// Mitsubishi GX Works2 project: BookEX6_47 Serial   PLC: Q13UDV

// global labels: Global
VAR_GLOBAL
  bVar0 AT M5000 : BOOL;
  abArray0 AT M5010 : ARRAY [0..49] OF BOOL;
  sStr0 AT D5000 : STRING[199];
  sStr1 AT D5100 : STRING[199];
  sStr2 AT D5200 : STRING[199];
  sStr3 AT D5300 : STRING[199];
  sStr4 AT D5400 : STRING[199];
  sStr5 AT D5500 : STRING[199];
  sStr6 AT D5600 : STRING[199];
  sStr7 AT D5700 : STRING[199];
  sStr8 AT D5800 : STRING[199];
  sStr9 AT D5900 : STRING[199];
  iVar0 AT D4500 : INT;
  iVar1 AT D4501 : INT;
  iVar2 AT D4502 : INT;
  iVar3 AT D4503 : INT;
  iVar4 AT D4504 : INT;
  iVar5 AT D4505 : INT;
  iVar6 AT D4506 : INT;
  iVar7 AT D4507 : INT;
  iVar8 AT D4508 : INT;
  iVar9 AT D4509 : INT;
  dVar0 AT D4510 : DINT;
  dVar1 AT D4512 : DINT;
  dVar2 AT D4514 : DINT;
  dVar3 AT D4516 : DINT;
  dVar4 AT D4518 : DINT;
  dVar5 AT D4520 : DINT;
  dVar6 AT D4522 : DINT;
  dVar7 AT D4524 : DINT;
  dVar8 AT D4526 : DINT;
  dVar9 AT D4528 : DINT;
  wVar0 AT D4530 : WORD;
  wVar1 AT D4531 : WORD;
  wVar2 AT D4532 : WORD;
  wVar3 AT D4533 : WORD;
  wVar4 AT D4534 : WORD;
  wVar5 AT D4535 : WORD;
  wVar6 AT D4536 : WORD;
  wVar7 AT D4537 : WORD;
  wVar8 AT D4538 : WORD;
  wVar9 AT D4539 : WORD;
  dwVar0 AT D4540 : DWORD;
  dwVar1 AT D4542 : DWORD;
  dwVar2 AT D4544 : DWORD;
  dwVar3 AT D4546 : DWORD;
  dwVar4 AT D4548 : DWORD;
  dwVar5 AT D4550 : DWORD;
  dwVar6 AT D4552 : DWORD;
  dwVar7 AT D4554 : DWORD;
  dwVar8 AT D4556 : DWORD;
  dwVar9 AT D4558 : DWORD;
  fsVar0 AT D4560 : REAL;
  fsVar1 AT D4562 : REAL;
  fsVar2 AT D4564 : REAL;
  fsVar3 AT D4566 : REAL;
  fsVar4 AT D4568 : REAL;
  fsVar5 AT D4570 : REAL;
  fsVar6 AT D4572 : REAL;
  fsVar7 AT D4574 : REAL;
  fsVar8 AT D4576 : REAL;
  fsVar9 AT D4578 : REAL;
  fdVar0 AT D4580 : LREAL;
  tTime0 AT D4620 : TIME;
  tTime1 AT D4622 : TIME;
  tTime2 AT D4624 : TIME;
  tTime3 AT D4626 : TIME;
  tTime4 AT D4628 : TIME;
  tTime5 AT D4630 : TIME;
  tTime6 AT D4632 : TIME;
  tTime7 AT D4634 : TIME;
  tTime8 AT D4636 : TIME;
  tTime9 AT D4638 : TIME;
  tTime10 AT D4640 : TIME;
  bVar1 AT M5001 : BOOL;
  bVar2 AT M5002 : BOOL;
  bVar3 AT M5003 : BOOL;
  bVar4 AT M5004 : BOOL;
  bVar5 AT M5005 : BOOL;
  bVar6 AT M5006 : BOOL;
  bVar7 AT M5007 : BOOL;
  bVar8 AT M5008 : BOOL;
  bVar9 AT M5009 : BOOL;
  abArray1 AT M5060 : ARRAY [0..49] OF BOOL;
  abArray2 AT M5110 : ARRAY [0..49] OF BOOL;
  abArray3 AT M5160 : ARRAY [0..49] OF BOOL;
  abArray4 AT M5210 : ARRAY [0..49] OF BOOL;
  abArray5 AT M5260 : ARRAY [0..49] OF BOOL;
  abArray6 AT M5310 : ARRAY [0..49] OF BOOL;
  abArray7 AT M5360 : ARRAY [0..49] OF BOOL;
  abArray8 AT M5410 : ARRAY [0..49] OF BOOL;
  abArray9 AT M5460 : ARRAY [0..49] OF BOOL;
  fdVar1 AT D4584 : LREAL;
  fdVar2 AT D4588 : LREAL;
  fdVar3 AT D4592 : LREAL;
  fdVar4 AT D4596 : LREAL;
  fdVar5 AT D4600 : LREAL;
  fdVar6 AT D4604 : LREAL;
  fdVar7 AT D4608 : LREAL;
  fdVar8 AT D4612 : LREAL;
  fdVar9 AT D4616 : LREAL;
  afsPen0 AT D2000 : ARRAY [0..499] OF REAL;
  afsPen1 AT D3000 : ARRAY [0..499] OF REAL;
  adwD10 AT D10 : ARRAY [0..9] OF DWORD;
  awD10 AT D10 : ARRAY [0..19] OF WORD;
  abM10 AT M10 : ARRAY [0..19] OF BOOL;
END_VAR

// global labels: CommVar
VAR_GLOBAL
  CommRx AT D100 : ARRAY [0..49] OF INT;
  CommTx AT D300 : ARRAY [0..49] OF INT;
  gbNormal AT M10 : BOOL;
  gbError AT M11 : BOOL;
  giErrCnt AT D12 : INT;
  giOKCnt AT D13 : INT;
END_VAR
// user libraries (not included): HMI

FUNCTION_BLOCK BattRequest
VAR_INPUT
  b_EN : BOOL;
END_VAR
VAR_OUTPUT
  b_ENO : BOOL;
END_VAR
VAR
  ix : INT;
  iy : INT;
  iz : INT;
END_VAR
;
b_ENO := b_EN;
IF b_EN THEN
	CommTX[0] := 11;
	CommTX[1] := HFAAF;
	CommTx[2] := H0560;
	CommTx[3] := H6001;
	CommTx[4] := H0047;
	CommTx[5] := HAF00;
	CommTx[6] := H00A0;
	iy := 0;
	FOR ix := 2 TO 4 DO
		iz := CommTx[ix] MOD 256;
		iy := iy + iz;
		iz := CommTx[ix] / 256;
		iy := iy + iz;
	END_FOR;
	CommTx[5] := CommTx[5] + (iy MOD 256);	
END_IF;
END_FUNCTION_BLOCK

FUNCTION_BLOCK BattStatus
VAR_INPUT
  b_EN : BOOL;
END_VAR
VAR_OUTPUT
  b_ENO : BOOL;
END_VAR
VAR
  ix : INT;
END_VAR
;
b_ENO := b_EN;
IF b_EN THEN
	ix := CommRx[4];
	SWAP(TRUE, ix);
	fsVar0 := INT_TO_REAL(ix) / 100.0;
	ix := CommRx[5];
	SWAP(TRUE, ix);
	fsVar1 := INT_TO_REAL(ix) / 100.0;
	ix := CommRx[6];
	SWAP(TRUE, ix);
	fsVar2 := INT_TO_REAL(ix);
	ix := CommRx[7];
	SWAP(TRUE, ix);
	fsVar3 := INT_TO_REAL(ix) / 10.0;
END_IF;
END_FUNCTION_BLOCK

PROGRAM ExBARCODE
(* structured ladder/FBD written out as ST: instructions are called as NAME(EN, inputs, outputs); _pN, _eN, _tN stand for wires *)
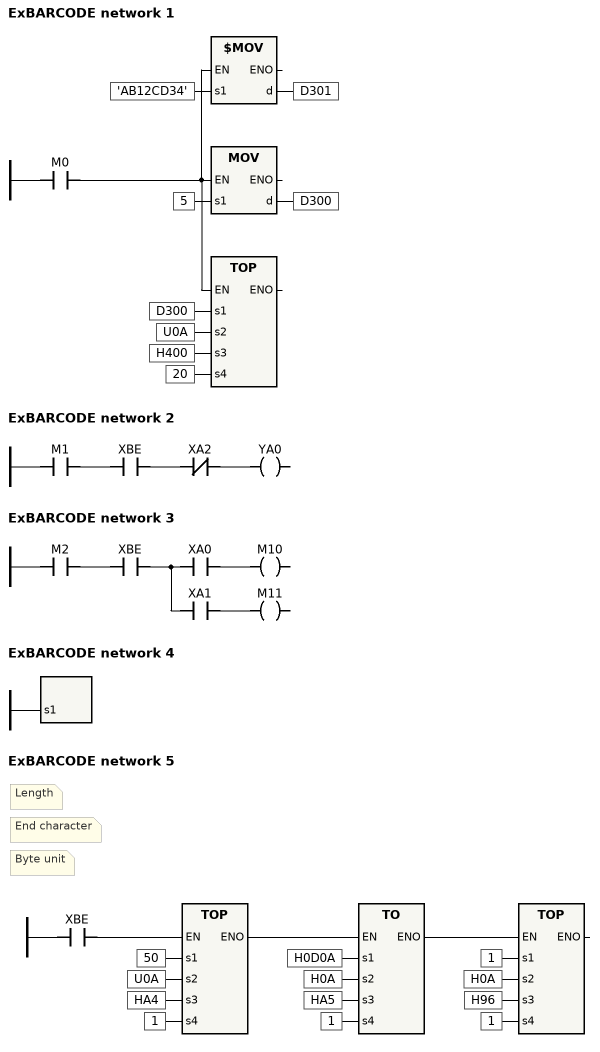
(* network 1 *)
$MOV(M0, 'AB12CD34', D301);
MOV(M0, 5, D300);
TOP(M0, D300, U0A, H400, 20);
(* network 2 *)
YA0 := M1 AND XBE AND NOT XA2;
(* network 3 *)
_p1 := M2 AND XBE;
M10 := _p1 AND XA0;
M11 := _p1 AND XA1;
(* network 4 *)
(* element kind 10  <- TRUE *)
(* network 5 *)
(* Length *)
(* End character *)
(* Byte unit *)
_e1 := TOP(XBE, 50, U0A, HA4, 1);
_e2 := TO(_e1, H0D0A, H0A, HA5, 1);
TOP(_e2, 1, H0A, H96, 1);
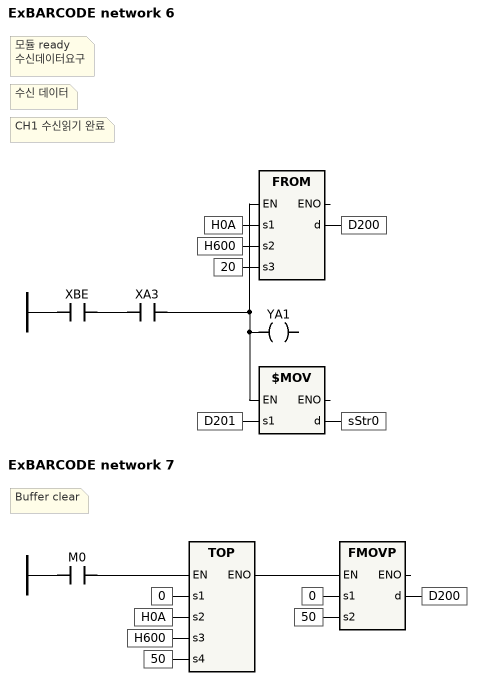
(* network 6 *)
(* 모듈 ready / 수신데이터요구 *)
(* 수신 데이터 *)
(* CH1 수신읽기 완료 *)
_p1 := XBE AND XA3;
FROM(_p1, H0A, H600, 20, D200);
YA1 := _p1;
$MOV(_p1, D201, sStr0);
(* network 7 *)
(* Buffer clear *)
_e1 := TOP(M0, 0, H0A, H600, 50);
FMOVP(_e1, 0, 50, D200);
END_PROGRAM

PROGRAM ExBIDIN
VAR
  aCtrlData : ARRAY [0..3] OF WORD;
  abComp : ARRAY [0..1] OF BOOL;
  bFlag : BOOL;
  bFlagExe : BOOL;
  bNormal : BOOL;
  bError : BOOL;
  Mov4WORD_1 : Mov4WORD;
  iErrCode : INT;
END_VAR
(* structured ladder/FBD written out as ST: instructions are called as NAME(EN, inputs, outputs); _pN, _eN, _tN stand for wires *)
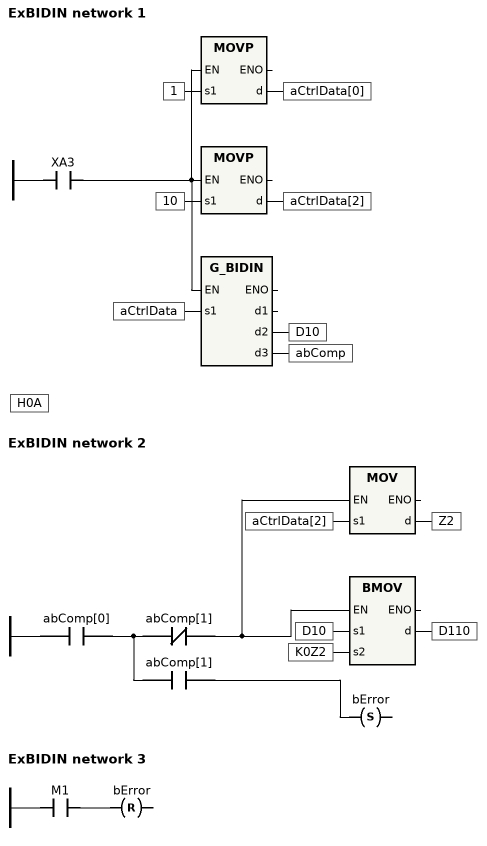
(* network 1 *)
MOVP(XA3, 1, aCtrlData[0]);
MOVP(XA3, 10, aCtrlData[2]);
G_BIDIN(XA3, aCtrlData, _open, D10, abComp);
(* not connected to any output: H0A *)
(* network 2 *)
_p1 := abComp[0] AND NOT abComp[1];
MOV(_p1, aCtrlData[2], Z2);
BMOV(_p1, D10, K0Z2, D110);
SET(abComp[0] AND abComp[1], bError);
(* network 3 *)
RST(M1, bError);
END_PROGRAM

PROGRAM ExBIDOUT
VAR
  aCtrlData : ARRAY [0..2] OF WORD;
  abComp : ARRAY [0..1] OF BOOL;
  bFlag : BOOL;
  bFlagExe : BOOL;
  bNormal : BOOL;
  bError : BOOL;
  Mov4WORD_1 : Mov4WORD;
  iErrCode : INT;
END_VAR
(* structured ladder/FBD written out as ST: instructions are called as NAME(EN, inputs, outputs); _pN, _eN, _tN stand for wires *)
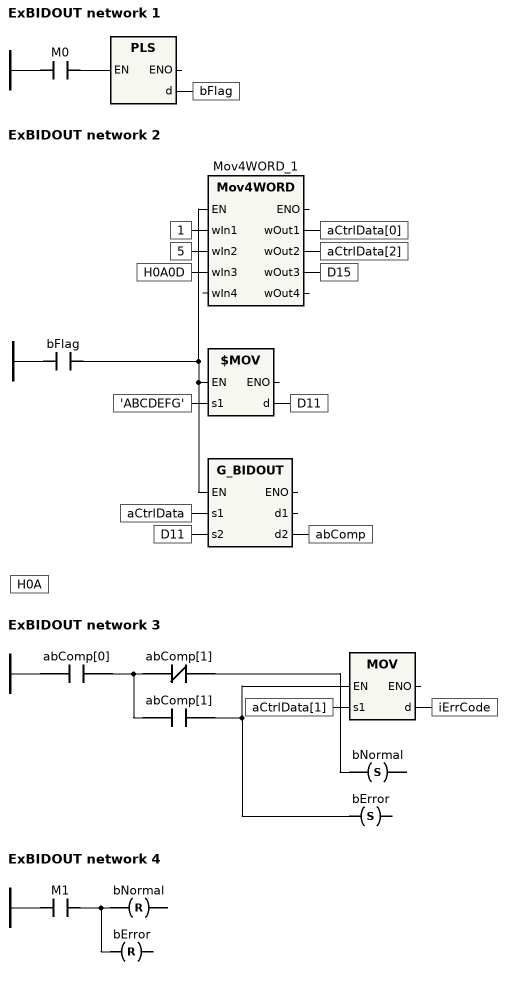
(* network 1 *)
PLS(M0, bFlag);
(* network 2 *)
Mov4WORD_1(EN := bFlag, wIn1 := 1, wIn2 := 5, wIn3 := H0A0D, wOut1 => aCtrlData[0], wOut2 => aCtrlData[2], wOut3 => D15);
$MOV(bFlag, 'ABCDEFG', D11);
G_BIDOUT(bFlag, aCtrlData, D11, _open, abComp);
(* not connected to any output: H0A *)
(* network 3 *)
SET(abComp[0] AND NOT abComp[1], bNormal);
_p1 := abComp[0] AND abComp[1];
MOV(_p1, aCtrlData[1], iErrCode);
SET(_p1, bError);
(* network 4 *)
RST(M1, bNormal);
RST(M1, bError);
END_PROGRAM

PROGRAM ExBUFRCVS_INT
VAR
  bNormal : BOOL;
  bError : BOOL;
  aCtrlTx : ARRAY [0..2] OF WORD;
  aCtrlRx : ARRAY [0..3] OF WORD;
  BattRequest_1 : BattRequest;
END_VAR
(* structured ladder/FBD written out as ST: instructions are called as NAME(EN, inputs, outputs); _pN, _eN, _tN stand for wires *)
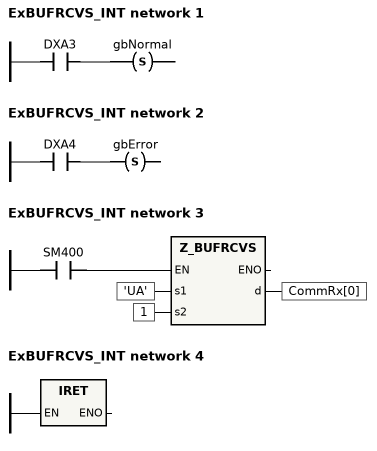
(* network 1 *)
SET(DXA3, gbNormal);
(* network 2 *)
SET(DXA4, gbError);
(* network 3 *)
Z_BUFRCVS(SM400, 'UA', 1, CommRx[0]);
(* network 4 *)
IRET(TRUE);
END_PROGRAM

PROGRAM ExBUFRCVS_MAIN
VAR
  aCtrlTx : ARRAY [0..2] OF WORD;
  aCtrlRx : ARRAY [0..3] OF WORD;
  BattRequest_1 : BattRequest;
  abComp : ARRAY [0..1] OF BOOL;
  BattStatus_1 : BattStatus;
END_VAR
(* structured ladder/FBD written out as ST: instructions are called as NAME(EN, inputs, outputs); _pN, _eN, _tN stand for wires *)
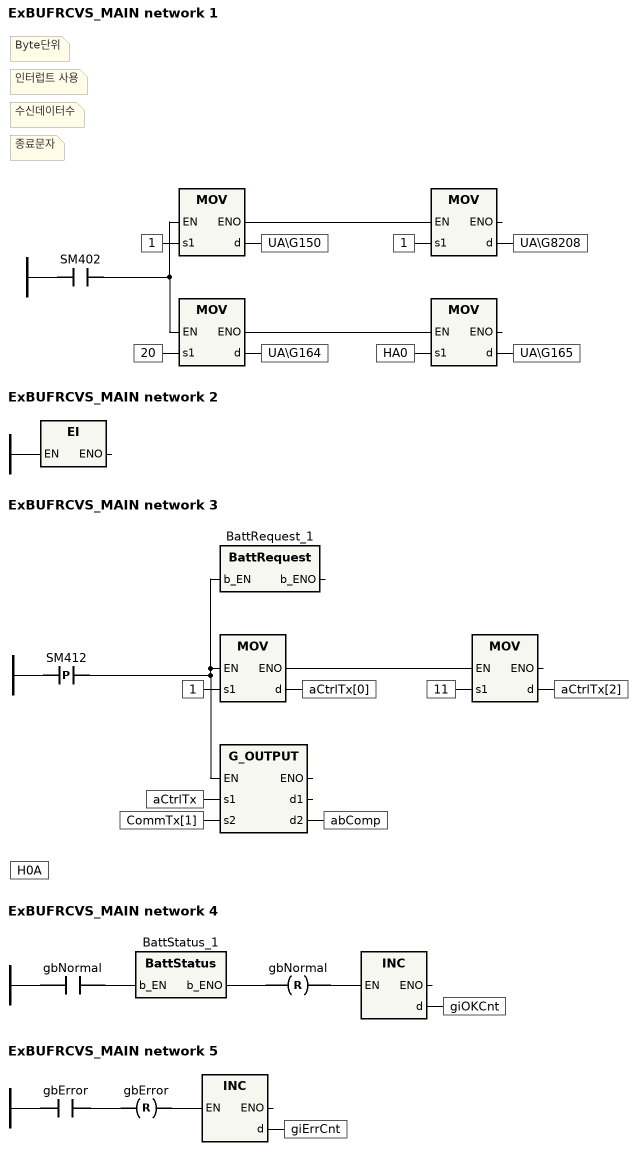
(* network 1 *)
(* Byte단위 *)
(* 인터럽트 사용 *)
(* 수신데이터수 *)
(* 종료문자 *)
_e1 := MOV(SM402, 1, UA\G150);
MOV(_e1, 1, UA\G8208);
_e2 := MOV(SM402, 20, UA\G164);
MOV(_e2, HA0, UA\G165);
(* network 2 *)
EI(TRUE);
(* network 3 *)
_p1 := LDP(TRUE, SM412);
BattRequest_1(b_EN := _p1);
_e2 := MOV(_p1, 1, aCtrlTx[0]);
MOV(_e2, 11, aCtrlTx[2]);
G_OUTPUT(_p1, aCtrlTx, CommTx[1], _open, abComp);
(* not connected to any output: H0A *)
(* network 4 *)
BattStatus_1(b_EN := gbNormal);
RST(BattStatus_1.b_ENO, gbNormal);
INC(BattStatus_1.b_ENO, giOKCnt);
(* network 5 *)
RST(gbError, gbError);
INC(gbError, giErrCnt);
END_PROGRAM

PROGRAM ExCPRTCL
VAR
  aCtrlData : ARRAY [0..17] OF WORD;
  abComp : ARRAY [0..1] OF BOOL;
  bFlag : BOOL;
  bFlagSet : BOOL;
  bFlagExe : BOOL;
  bNormal : BOOL;
  bError : BOOL;
  Mov4WORD_1 : Mov4WORD;
  iErrCode : INT;
  Mov8WORD_1 : Mov8WORD;
  Mov8WORD_2 : Mov8WORD;
  Mov8WORD_3 : Mov8WORD;
  BattRequest_1 : BattRequest;
  BattStatus_1 : BattStatus;
END_VAR
(* structured ladder/FBD written out as ST: instructions are called as NAME(EN, inputs, outputs); _pN, _eN, _tN stand for wires *)
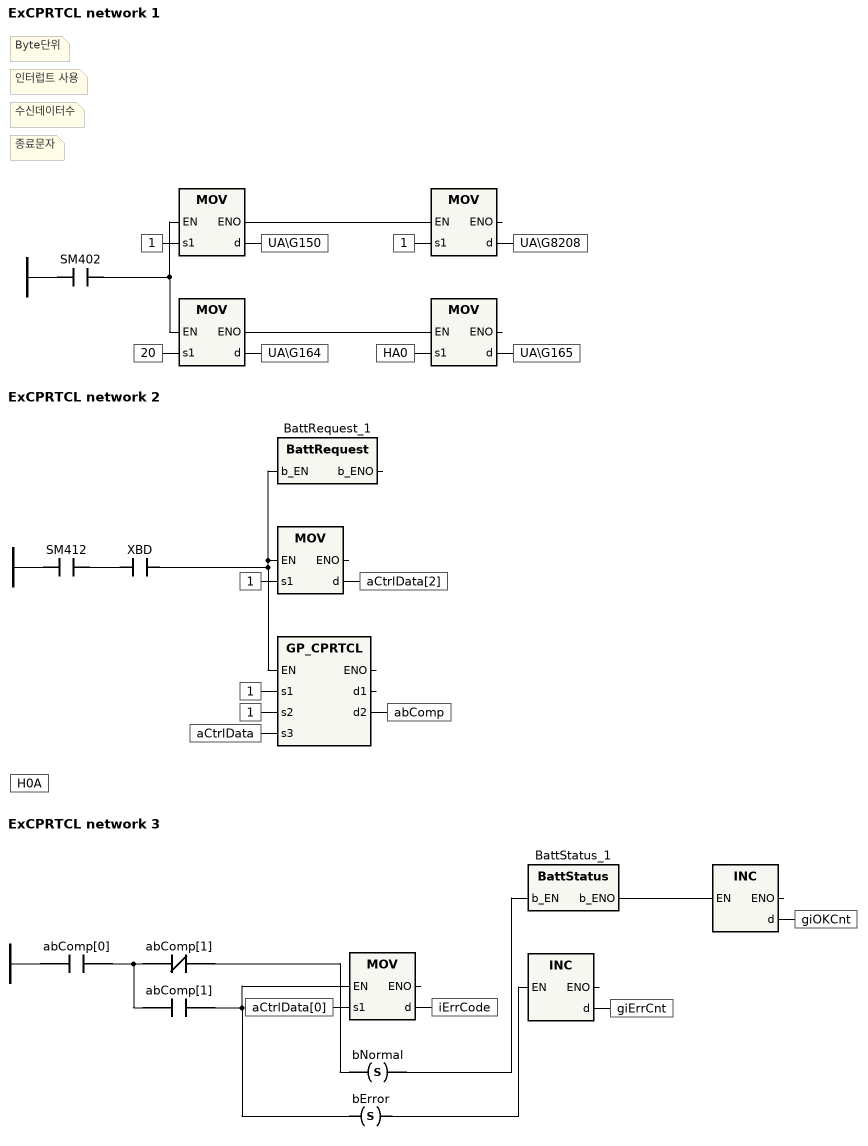
(* network 1 *)
(* Byte단위 *)
(* 인터럽트 사용 *)
(* 수신데이터수 *)
(* 종료문자 *)
_e1 := MOV(SM402, 1, UA\G150);
MOV(_e1, 1, UA\G8208);
_e2 := MOV(SM402, 20, UA\G164);
MOV(_e2, HA0, UA\G165);
(* network 2 *)
_p1 := SM412 AND XBD;
BattRequest_1(b_EN := _p1);
MOV(_p1, 1, aCtrlData[2]);
GP_CPRTCL(_p1, 1, 1, aCtrlData, _open, abComp);
(* not connected to any output: H0A *)
(* network 3 *)
_p1 := abComp[0] AND NOT abComp[1];
SET(_p1, bNormal);
BattStatus_1(b_EN := _p1);
INC(BattStatus_1.b_ENO, giOKCnt);
_p2 := abComp[0] AND abComp[1];
SET(_p2, bError);
INC(_p2, giErrCnt);
MOV(_p2, aCtrlData[0], iErrCode);
END_PROGRAM

PROGRAM ExCSET
VAR
  aCtrlData : ARRAY [0..111] OF WORD;
  abComp : ARRAY [0..1] OF BOOL;
  bFlag2 : BOOL;
  bFlagExe2 : BOOL;
  bNormal : BOOL;
  bError : BOOL;
  Mov4WORD_1 : Mov4WORD;
  iErrCode : INT;
  Mov8WORD_1 : Mov8WORD;
  bFlagSet2 : BOOL;
  Mov8WORD_2 : Mov8WORD;
  Mov8WORD_3 : Mov8WORD;
  Dummy : INT;
  bFlag3 : BOOL;
  bFlagSet3 : BOOL;
  bFlagExe3 : BOOL;
END_VAR
(* structured ladder/FBD written out as ST: instructions are called as NAME(EN, inputs, outputs); _pN, _eN, _tN stand for wires *)
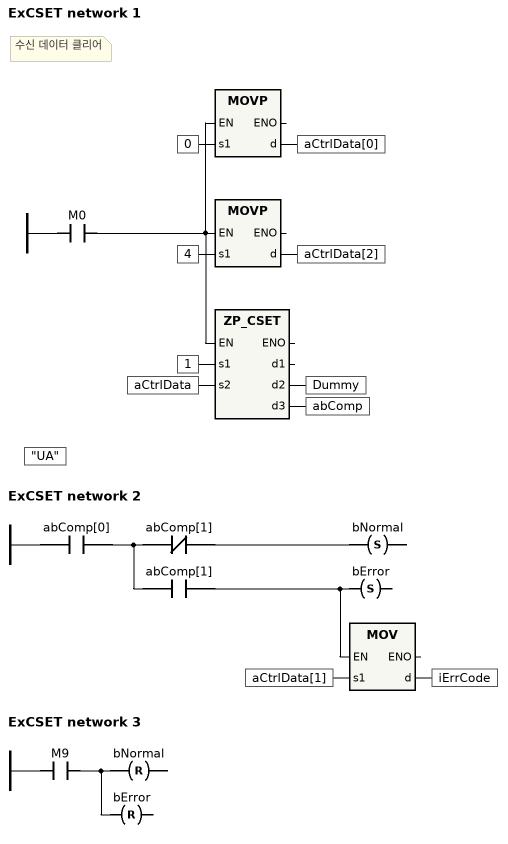
(* network 1 *)
(* 수신 데이터 클리어 *)
MOVP(M0, 0, aCtrlData[0]);
MOVP(M0, 4, aCtrlData[2]);
ZP_CSET(M0, 1, aCtrlData, _open, Dummy, abComp);
(* not connected to any output: "UA" *)
(* network 2 *)
SET(abComp[0] AND NOT abComp[1], bNormal);
_p1 := abComp[0] AND abComp[1];
SET(_p1, bError);
MOV(_p1, aCtrlData[1], iErrCode);
(* network 3 *)
RST(M9, bNormal);
RST(M9, bError);
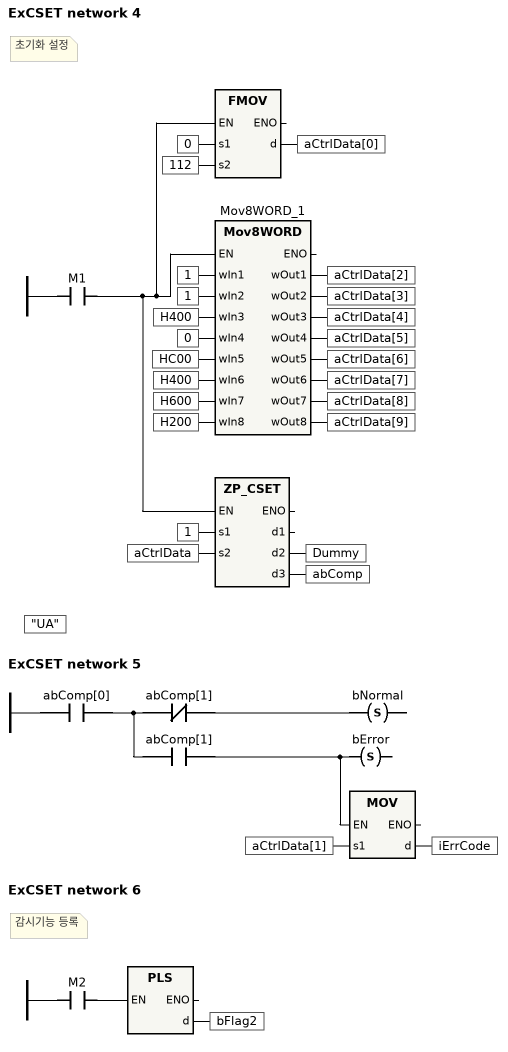
(* network 4 *)
(* 초기화 설정 *)
FMOV(M1, 0, 112, aCtrlData[0]);
Mov8WORD_1(EN := M1, wIn1 := 1, wIn2 := 1, wIn3 := H400, wIn4 := 0, wIn5 := HC00, wIn6 := H400, wIn7 := H600, wIn8 := H200, wOut1 => aCtrlData[2], wOut2 => aCtrlData[3], wOut3 => aCtrlData[4], wOut4 => aCtrlData[5], wOut5 => aCtrlData[6], wOut6 => aCtrlData[7], wOut7 => aCtrlData[8], wOut8 => aCtrlData[9]);
ZP_CSET(M1, 1, aCtrlData, _open, Dummy, abComp);
(* not connected to any output: "UA" *)
(* network 5 *)
SET(abComp[0] AND NOT abComp[1], bNormal);
_p1 := abComp[0] AND abComp[1];
SET(_p1, bError);
MOV(_p1, aCtrlData[1], iErrCode);
(* network 6 *)
(* 감시기능 등록 *)
PLS(M2, bFlag2);
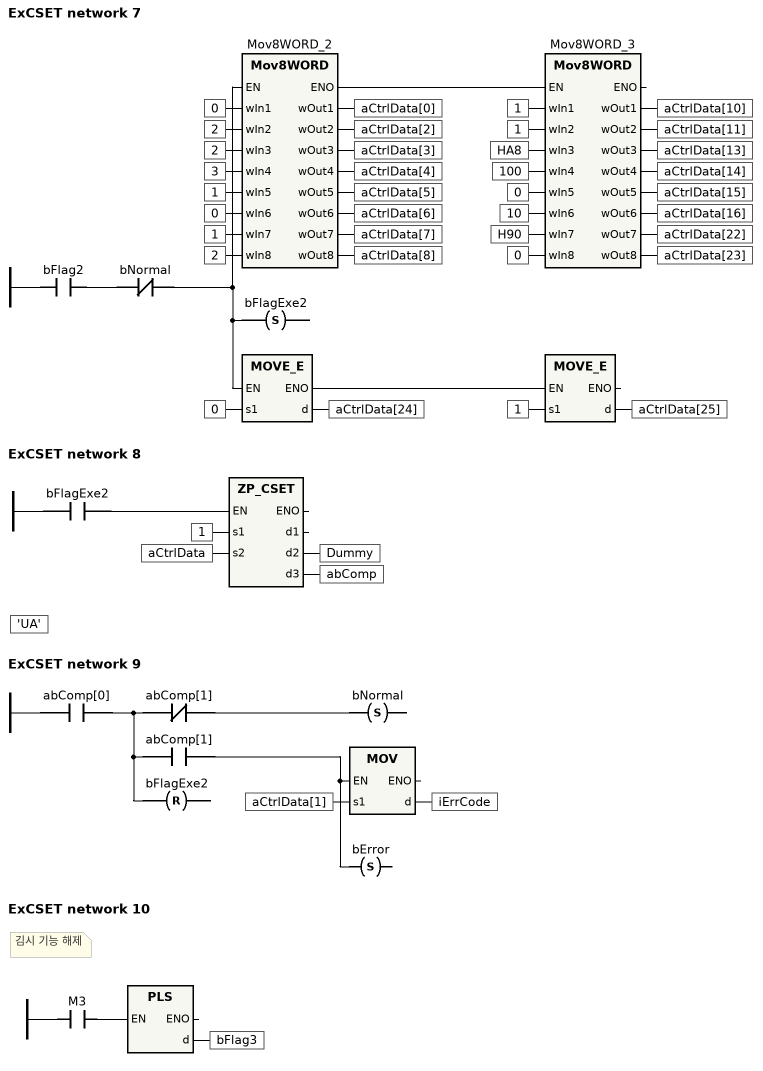
(* network 7 *)
_p1 := bFlag2 AND NOT bNormal;
Mov8WORD_2(EN := _p1, wIn1 := 0, wIn2 := 2, wIn3 := 2, wIn4 := 3, wIn5 := 1, wIn6 := 0, wIn7 := 1, wIn8 := 2, wOut1 => aCtrlData[0], wOut2 => aCtrlData[2], wOut3 => aCtrlData[3], wOut4 => aCtrlData[4], wOut5 => aCtrlData[5], wOut6 => aCtrlData[6], wOut7 => aCtrlData[7], wOut8 => aCtrlData[8]);
Mov8WORD_3(EN := Mov8WORD_2.ENO, wIn1 := 1, wIn2 := 1, wIn3 := HA8, wIn4 := 100, wIn5 := 0, wIn6 := 10, wIn7 := H90, wIn8 := 0, wOut1 => aCtrlData[10], wOut2 => aCtrlData[11], wOut3 => aCtrlData[13], wOut4 => aCtrlData[14], wOut5 => aCtrlData[15], wOut6 => aCtrlData[16], wOut7 => aCtrlData[22], wOut8 => aCtrlData[23]);
_e2 := MOVE_E(_p1, 0, aCtrlData[24]);
MOVE_E(_e2, 1, aCtrlData[25]);
SET(_p1, bFlagExe2);
(* network 8 *)
ZP_CSET(bFlagExe2, 1, aCtrlData, _open, Dummy, abComp);
(* not connected to any output: 'UA' *)
(* network 9 *)
SET(abComp[0] AND NOT abComp[1], bNormal);
_p1 := abComp[0] AND abComp[1];
SET(_p1, bError);
MOV(_p1, aCtrlData[1], iErrCode);
RST(abComp[0], bFlagExe2);
(* network 10 *)
(* 김시 기능 해제 *)
PLS(M3, bFlag3);
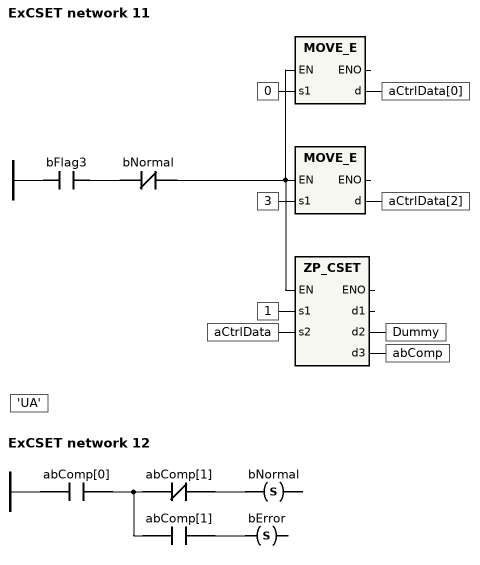
(* network 11 *)
_p1 := bFlag3 AND NOT bNormal;
MOVE_E(_p1, 0, aCtrlData[0]);
MOVE_E(_p1, 3, aCtrlData[2]);
ZP_CSET(_p1, 1, aCtrlData, _open, Dummy, abComp);
(* not connected to any output: 'UA' *)
(* network 12 *)
SET(abComp[0] AND NOT abComp[1], bNormal);
SET(abComp[0] AND abComp[1], bError);
END_PROGRAM

PROGRAM ExGETE
VAR
  aCtrlData : ARRAY [0..3] OF WORD;
  abComp : ARRAY [0..1] OF BOOL;
  bFlag : BOOL;
  bFlagSet : BOOL;
  bFlagExe : BOOL;
  bNormal : BOOL;
  bError : BOOL;
  Mov4WORD_1 : Mov4WORD;
  iErrCode : INT;
  Mov8WORD_1 : Mov8WORD;
  Mov8WORD_2 : Mov8WORD;
  Mov8WORD_3 : Mov8WORD;
  aFrame : ARRAY [0..99] OF WORD;
  abComp1 : ARRAY [0..1] OF BOOL;
END_VAR
(* structured ladder/FBD written out as ST: instructions are called as NAME(EN, inputs, outputs); _pN, _eN, _tN stand for wires *)
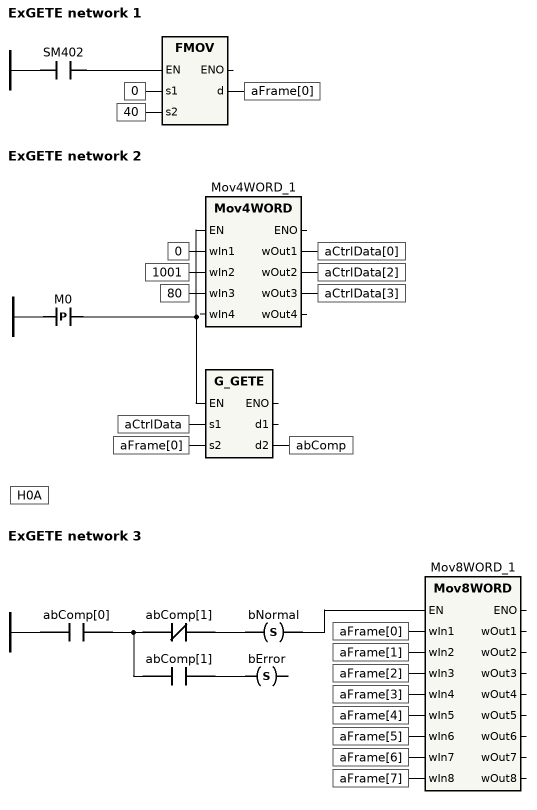
(* network 1 *)
FMOV(SM402, 0, 40, aFrame[0]);
(* network 2 *)
_p1 := LDP(TRUE, M0);
Mov4WORD_1(EN := _p1, wIn1 := 0, wIn2 := 1001, wIn3 := 80, wOut1 => aCtrlData[0], wOut2 => aCtrlData[2], wOut3 => aCtrlData[3]);
G_GETE(_p1, aCtrlData, aFrame[0], _open, abComp);
(* not connected to any output: H0A *)
(* network 3 *)
_p1 := abComp[0] AND NOT abComp[1];
SET(_p1, bNormal);
Mov8WORD_1(EN := _p1, wIn1 := aFrame[0], wIn2 := aFrame[1], wIn3 := aFrame[2], wIn4 := aFrame[3], wIn5 := aFrame[4], wIn6 := aFrame[5], wIn7 := aFrame[6], wIn8 := aFrame[7]);
SET(abComp[0] AND abComp[1], bError);
END_PROGRAM

PROGRAM ExIN_OUT
VAR
  aCtrlTx : ARRAY [0..2] OF WORD;
  ix : INT;
  iy : INT;
  iz : INT;
  wx : WORD;
  wBuff : ARRAY [0..9] OF WORD;
  aCtrlRx : ARRAY [0..3] OF WORD;
  abComp1 : ARRAY [0..1] OF BOOL;
  abComp2 : ARRAY [0..1] OF BOOL;
  fbBattRequest : BattRequest;
  fbBattStatus : BattStatus;
END_VAR
;
IF SM402 THEN
	TO(TRUE, 1, H0A, H96, 1);
	wBuff[0] := 20;
	wBuff[1] := HA0;
	TO(TRUE, wBuff[0], H0A, HA4, 2);
END_IF;  
IF LDP(TRUE, SM412) THEN
	fbBattRequest(b_EN := TRUE);
	aCtrlTx[0] := 1;
	aCtrlTx[2] := 11;
	G_OUTPUT(TRUE, H0A, aCtrlTx, CommTx[1], abComp1);
END_IF;
IF XBE AND  XA3 THEN
	aCtrlRx[0] := 1;
	aCtrlRx[3] := 17;
	G_INPUT(TRUE, H0A, aCtrlRx, CommRx[1], abComp2);
END_IF;
IF abComp2[0] AND NOT abComp2[1] THEN
	fbBattStatus(b_EN := TRUE);
END_IF;
END_PROGRAM

PROGRAM ExINPUT
VAR
  abComp : ARRAY [0..1] OF BOOL;
  bFlag : BOOL;
  bFlagExe : BOOL;
  bNormal : BOOL;
  bError : BOOL;
  Mov4WORD_1 : Mov4WORD;
  aCtrlData : ARRAY [0..3] OF WORD;
END_VAR
(* structured ladder/FBD written out as ST: instructions are called as NAME(EN, inputs, outputs); _pN, _eN, _tN stand for wires *)
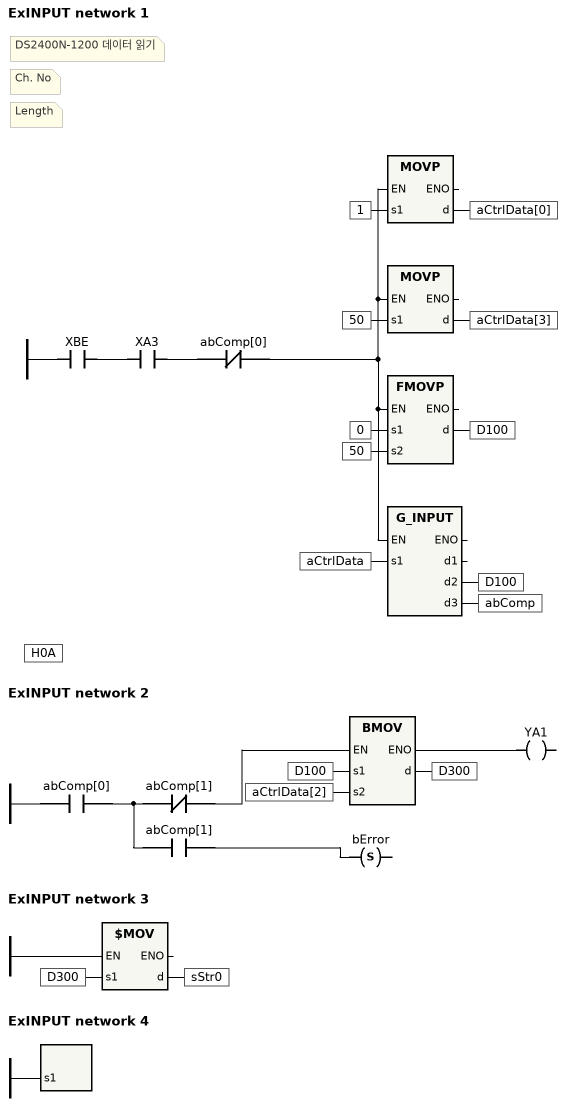
(* network 1 *)
(* DS2400N-1200 데이터 읽기 *)
(* Ch. No *)
(* Length *)
_p1 := XBE AND XA3 AND NOT abComp[0];
MOVP(_p1, 1, aCtrlData[0]);
MOVP(_p1, 50, aCtrlData[3]);
FMOVP(_p1, 0, 50, D100);
G_INPUT(_p1, aCtrlData, _open, D100, abComp);
(* not connected to any output: H0A *)
(* network 2 *)
_e1 := BMOV(abComp[0] AND NOT abComp[1], D100, aCtrlData[2], D300);
YA1 := _e1;
SET(abComp[0] AND abComp[1], bError);
(* network 3 *)
$MOV(TRUE, D300, sStr0);
(* network 4 *)
(* element kind 10  <- TRUE *)
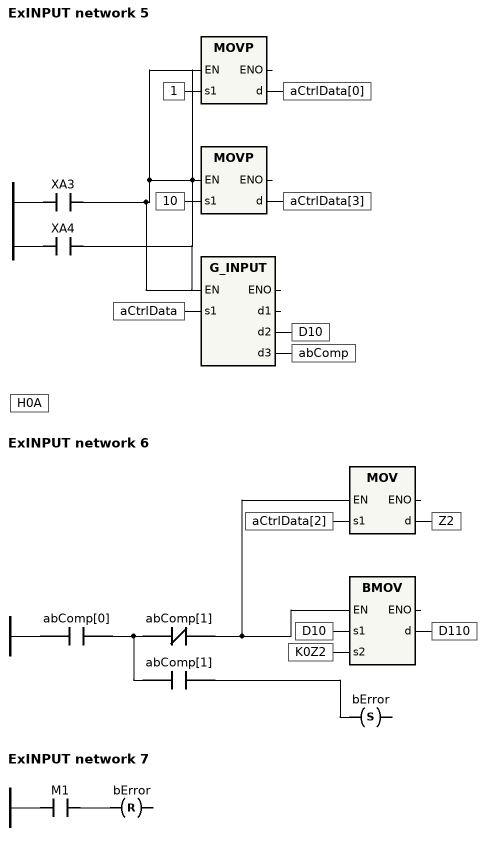
(* network 5 *)
_p1 := XA3 OR XA4;
MOVP(_p1, 1, aCtrlData[0]);
MOVP(_p1, 10, aCtrlData[3]);
G_INPUT(_p1, aCtrlData, _open, D10, abComp);
(* not connected to any output: H0A *)
(* network 6 *)
_p1 := abComp[0] AND NOT abComp[1];
MOV(_p1, aCtrlData[2], Z2);
BMOV(_p1, D10, K0Z2, D110);
SET(abComp[0] AND abComp[1], bError);
(* network 7 *)
RST(M1, bError);
END_PROGRAM

PROGRAM ExNoINST
VAR
  ix : INT;
  iy : INT;
  iz : INT;
  wx : WORD;
  wBuff : ARRAY [0..9] OF WORD;
  fbBattRequest : BattRequest;
  fbBattStatus : BattStatus;
END_VAR
;
;(*
;        Communication with Battery             ;
;				TX Format		RX Format
; 0xAF	STX1					0xAF	
; 0xFA	STX2            		0xFA	
; 0x60		Address         	0x60	
; 0x05		Length          		0x0B	or 0x07 (error)
; 0x01		Command       0x03	or 0x1F (error)	
; 0x60		Order           		0x60	
; 0x47		Data1           		...	Datahi Datalow 4set	
; 0x00		Data2           		...	
; 0x0D	Checksum       0x??	
; 0xAF	ETX1            		0xAF	
; 0xA0 	ETX2            		0xA0    
*)
IF SM402 THEN
	TO(TRUE, 1, H0A, H96, 1);
 	wBuff[0] := 20;
	wBuff[1] := HA0;   
(*	wBuff[0] := 17;
	wBuff[1] := HFFFF;  *)
	TO(TRUE, wBuff[0], H0A, HA4, 2);
END_IF;

IF LDP(TRUE, SM412) THEN
	fbBattRequest(b_EN := TRUE);
	TO(TRUE, CommTx[0], H0A, H400, 7);
	YA0 := TRUE;
	TO(TRUE, 0, H0A, H600, 20);
END_IF;
IF XA0 OR XA1 THEN
	YA0 := FALSE;
END_IF;

IF XBE AND  XA3 THEN
	FROM(TRUE, H0A, H600, 10,  CommRx[0]); 
	fbBattStatus(b_EN := TRUE);
	YA1 := TRUE;
END_IF;
IF NOT XBE OR NOT XA3 THEN
	YA1 := FALSE;
END_IF;
END_PROGRAM

PROGRAM ExONDEMAND
VAR
  aCtrlData : ARRAY [0..2] OF WORD;
  abComp : ARRAY [0..1] OF BOOL;
  bFlag : BOOL;
  bFlagExe : BOOL;
  Mov4WORD_1 : Mov4WORD;
  bNormal : BOOL;
  bError : BOOL;
END_VAR
(* structured ladder/FBD written out as ST: instructions are called as NAME(EN, inputs, outputs); _pN, _eN, _tN stand for wires *)
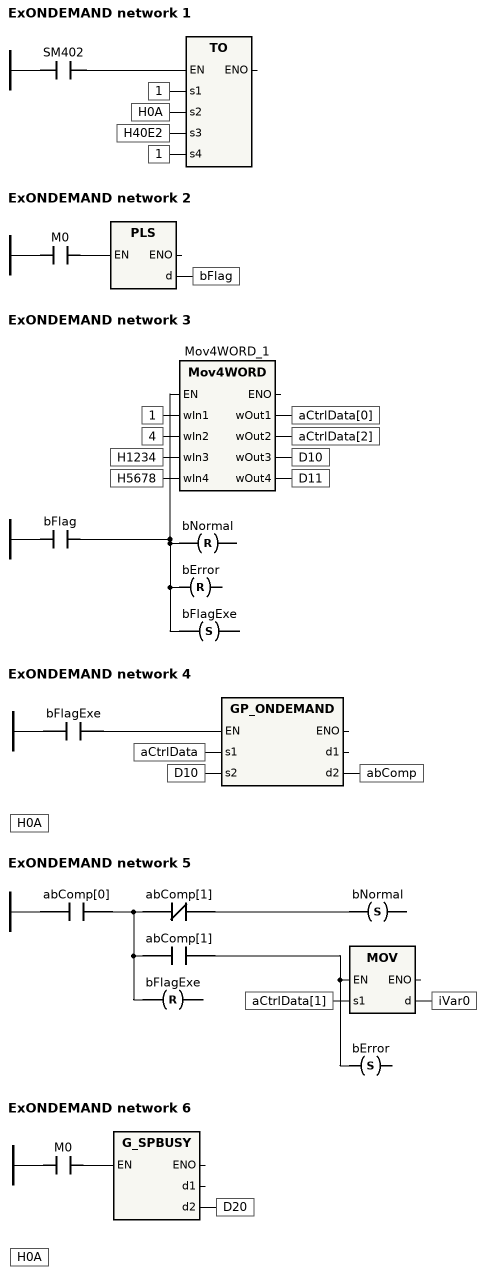
(* network 1 *)
TO(SM402, 1, H0A, H40E2, 1);
(* network 2 *)
PLS(M0, bFlag);
(* network 3 *)
Mov4WORD_1(EN := bFlag, wIn1 := 1, wIn2 := 4, wIn3 := H1234, wIn4 := H5678, wOut1 => aCtrlData[0], wOut2 => aCtrlData[2], wOut3 => D10, wOut4 => D11);
RST(bFlag, bNormal);
RST(bFlag, bError);
SET(bFlag, bFlagExe);
(* network 4 *)
GP_ONDEMAND(bFlagExe, aCtrlData, D10, _open, abComp);
(* not connected to any output: H0A *)
(* network 5 *)
SET(abComp[0] AND NOT abComp[1], bNormal);
_p1 := abComp[0] AND abComp[1];
SET(_p1, bError);
RST(abComp[0], bFlagExe);
MOV(_p1, aCtrlData[1], iVar0);
(* network 6 *)
G_SPBUSY(M0, _open, D20);
(* not connected to any output: H0A *)
END_PROGRAM

PROGRAM ExOUTPUT
VAR
  aCtrlData : ARRAY [0..2] OF WORD;
  abComp : ARRAY [0..1] OF BOOL;
  bFlag : BOOL;
  bFlagExe : BOOL;
  bNormal : BOOL;
  bError : BOOL;
  Mov4WORD_1 : Mov4WORD;
  iErrCode : INT;
  Mov8INT_1 : Mov8INT;
END_VAR
(* structured ladder/FBD written out as ST: instructions are called as NAME(EN, inputs, outputs); _pN, _eN, _tN stand for wires *)
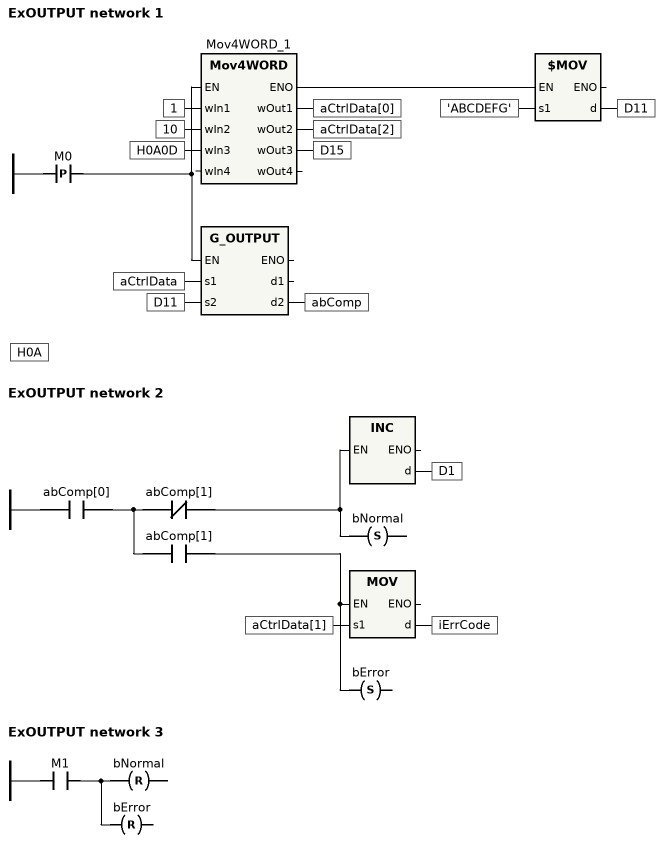
(* network 1 *)
_p1 := LDP(TRUE, M0);
Mov4WORD_1(EN := _p1, wIn1 := 1, wIn2 := 10, wIn3 := H0A0D, wOut1 => aCtrlData[0], wOut2 => aCtrlData[2], wOut3 => D15);
$MOV(Mov4WORD_1.ENO, 'ABCDEFG', D11);
G_OUTPUT(_p1, aCtrlData, D11, _open, abComp);
(* not connected to any output: H0A *)
(* network 2 *)
_p1 := abComp[0] AND NOT abComp[1];
SET(_p1, bNormal);
INC(_p1, D1);
_p2 := abComp[0] AND abComp[1];
MOV(_p2, aCtrlData[1], iErrCode);
SET(_p2, bError);
(* network 3 *)
RST(M1, bNormal);
RST(M1, bError);
END_PROGRAM

PROGRAM ExPRR
VAR
  aCtrlData : ARRAY [0..4] OF WORD;
  abComp : ARRAY [0..1] OF BOOL;
  bFlag : BOOL;
  bFlagExe : BOOL;
  bNormal : BOOL;
  bError : BOOL;
  Mov4WORD_1 : Mov4WORD;
  iErrCode : INT;
  Mov4WORD_2 : Mov4WORD;
  Mov4WORD_3 : Mov4WORD;
  Mov8WORD_1 : Mov8WORD;
  aFrame : ARRAY [0..5] OF WORD;
  aSendData : ARRAY [0..9] OF WORD;
  BattRequest_1 : BattRequest;
  BattStatus_1 : BattStatus;
  Mov8WORD_2 : Mov8WORD;
  aCtrlRx : ARRAY [0..3] OF WORD;
  abCompInst : ARRAY [0..1] OF BOOL;
END_VAR
(* structured ladder/FBD written out as ST: instructions are called as NAME(EN, inputs, outputs); _pN, _eN, _tN stand for wires *)
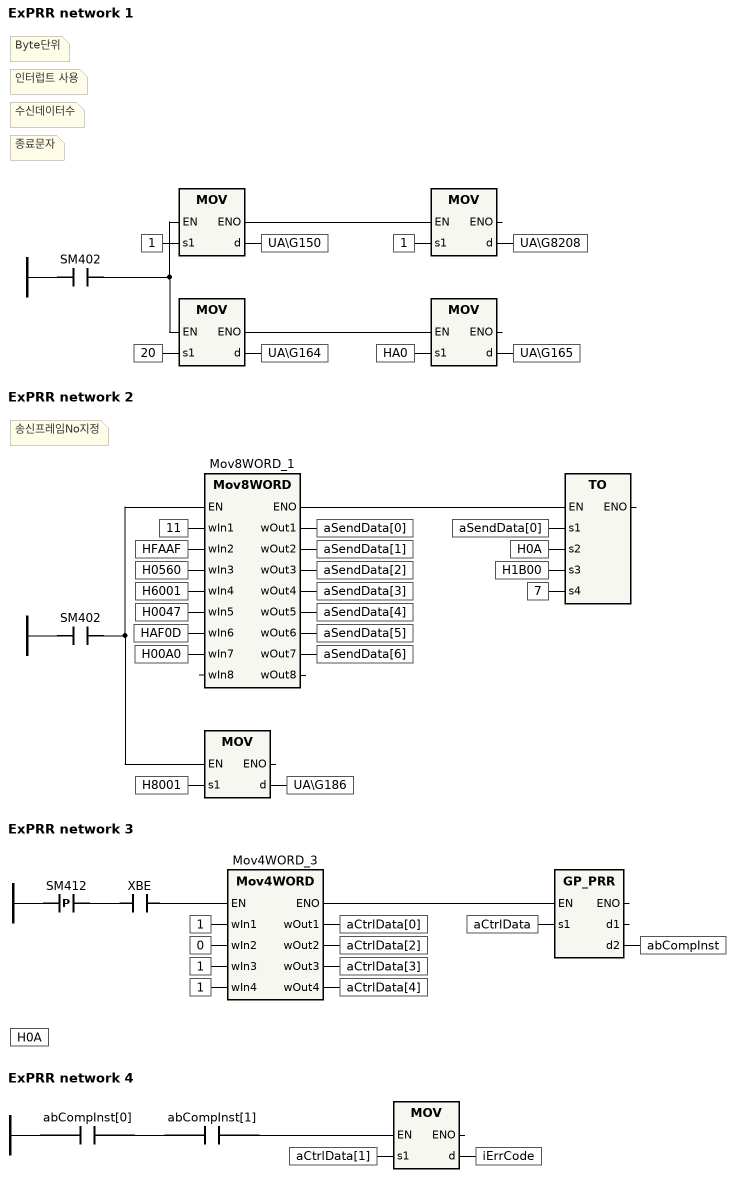
(* network 1 *)
(* Byte단위 *)
(* 인터럽트 사용 *)
(* 수신데이터수 *)
(* 종료문자 *)
_e1 := MOV(SM402, 1, UA\G150);
MOV(_e1, 1, UA\G8208);
_e2 := MOV(SM402, 20, UA\G164);
MOV(_e2, HA0, UA\G165);
(* network 2 *)
(* 송신프레임No지정 *)
Mov8WORD_1(EN := SM402, wIn1 := 11, wIn2 := HFAAF, wIn3 := H0560, wIn4 := H6001, wIn5 := H0047, wIn6 := HAF0D, wIn7 := H00A0, wOut1 => aSendData[0], wOut2 => aSendData[1], wOut3 => aSendData[2], wOut4 => aSendData[3], wOut5 => aSendData[4], wOut6 => aSendData[5], wOut7 => aSendData[6]);
TO(Mov8WORD_1.ENO, aSendData[0], H0A, H1B00, 7);
MOV(SM402, H8001, UA\G186);
(* network 3 *)
Mov4WORD_3(EN := LDP(TRUE, SM412) AND XBE, wIn1 := 1, wIn2 := 0, wIn3 := 1, wIn4 := 1, wOut1 => aCtrlData[0], wOut2 => aCtrlData[2], wOut3 => aCtrlData[3], wOut4 => aCtrlData[4]);
GP_PRR(Mov4WORD_3.ENO, aCtrlData, _open, abCompInst);
(* not connected to any output: H0A *)
(* network 4 *)
MOV(abCompInst[0] AND abCompInst[1], aCtrlData[1], iErrCode);
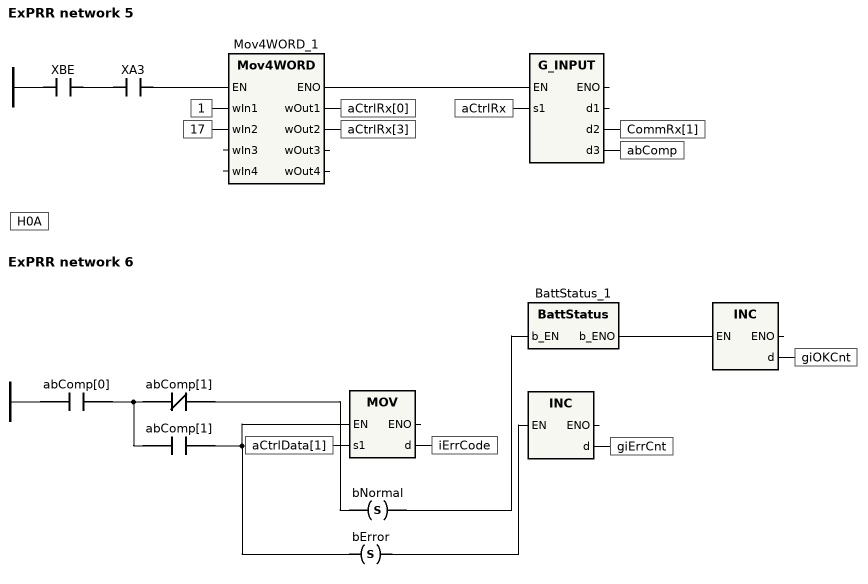
(* network 5 *)
Mov4WORD_1(EN := XBE AND XA3, wIn1 := 1, wIn2 := 17, wOut1 => aCtrlRx[0], wOut2 => aCtrlRx[3]);
G_INPUT(Mov4WORD_1.ENO, aCtrlRx, _open, CommRx[1], abComp);
(* not connected to any output: H0A *)
(* network 6 *)
_p1 := abComp[0] AND NOT abComp[1];
SET(_p1, bNormal);
BattStatus_1(b_EN := _p1);
INC(BattStatus_1.b_ENO, giOKCnt);
_p2 := abComp[0] AND abComp[1];
SET(_p2, bError);
INC(_p2, giErrCnt);
MOV(_p2, aCtrlData[1], iErrCode);
END_PROGRAM

PROGRAM ExPUTE
VAR
  aCtrlData : ARRAY [0..3] OF WORD;
  abComp : ARRAY [0..1] OF BOOL;
  bFlag : BOOL;
  bFlagSet : BOOL;
  bFlagExe : BOOL;
  bNormal : BOOL;
  bError : BOOL;
  Mov4WORD_1 : Mov4WORD;
  iErrCode : INT;
  Mov8WORD_1 : Mov8WORD;
  Mov8WORD_2 : Mov8WORD;
  Mov8WORD_3 : Mov8WORD;
  aFrame : ARRAY [0..99] OF WORD;
  abComp1 : ARRAY [0..1] OF BOOL;
END_VAR
(* structured ladder/FBD written out as ST: instructions are called as NAME(EN, inputs, outputs); _pN, _eN, _tN stand for wires *)
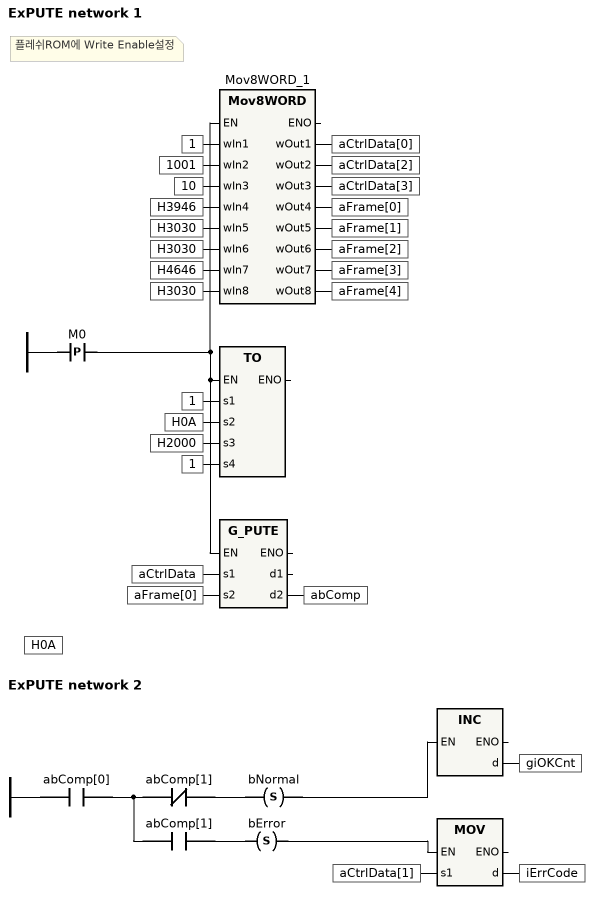
(* network 1 *)
(* 플레쉬ROM에 Write Enable설정 *)
_p1 := LDP(TRUE, M0);
Mov8WORD_1(EN := _p1, wIn1 := 1, wIn2 := 1001, wIn3 := 10, wIn4 := H3946, wIn5 := H3030, wIn6 := H3030, wIn7 := H4646, wIn8 := H3030, wOut1 => aCtrlData[0], wOut2 => aCtrlData[2], wOut3 => aCtrlData[3], wOut4 => aFrame[0], wOut5 => aFrame[1], wOut6 => aFrame[2], wOut7 => aFrame[3], wOut8 => aFrame[4]);
TO(_p1, 1, H0A, H2000, 1);
G_PUTE(_p1, aCtrlData, aFrame[0], _open, abComp);
(* not connected to any output: H0A *)
(* network 2 *)
_p1 := abComp[0] AND NOT abComp[1];
SET(_p1, bNormal);
INC(_p1, giOKCnt);
_p2 := abComp[0] AND abComp[1];
SET(_p2, bError);
MOV(_p2, aCtrlData[1], iErrCode);
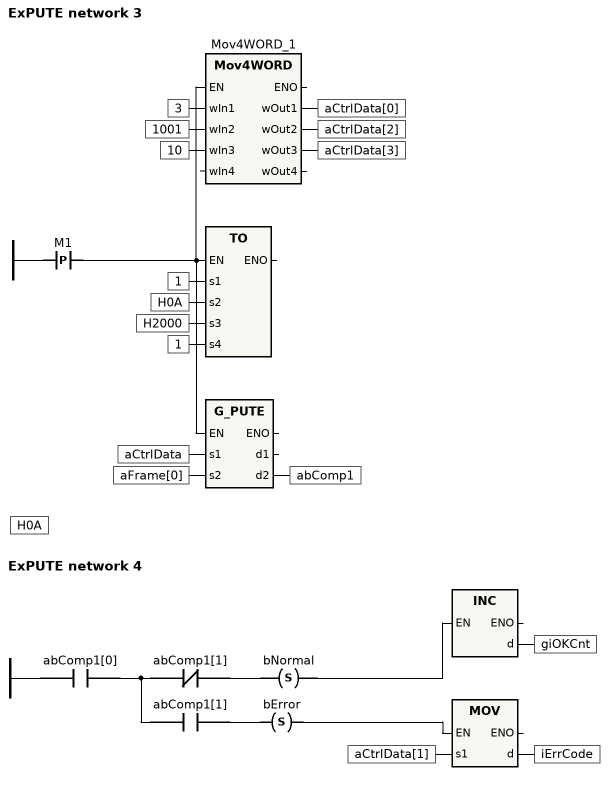
(* network 3 *)
_p1 := LDP(TRUE, M1);
Mov4WORD_1(EN := _p1, wIn1 := 3, wIn2 := 1001, wIn3 := 10, wOut1 => aCtrlData[0], wOut2 => aCtrlData[2], wOut3 => aCtrlData[3]);
TO(_p1, 1, H0A, H2000, 1);
G_PUTE(_p1, aCtrlData, aFrame[0], _open, abComp1);
(* not connected to any output: H0A *)
(* network 4 *)
_p1 := abComp1[0] AND NOT abComp1[1];
SET(_p1, bNormal);
INC(_p1, giOKCnt);
_p2 := abComp1[0] AND abComp1[1];
SET(_p2, bError);
MOV(_p2, aCtrlData[1], iErrCode);
END_PROGRAM

PROGRAM ExSPBUSY
(* structured ladder/FBD written out as ST: instructions are called as NAME(EN, inputs, outputs); _pN, _eN, _tN stand for wires *)
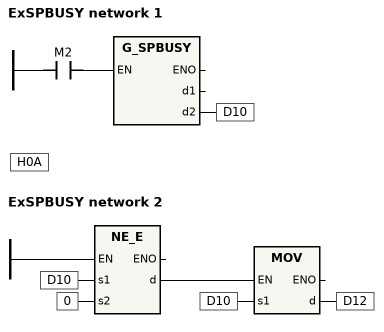
(* network 1 *)
G_SPBUSY(M2, _open, D10);
(* not connected to any output: H0A *)
(* network 2 *)
NE_E(TRUE, D10, 0, _t1);
MOV(_t1, D10, D12);
END_PROGRAM

PROGRAM ExUINI
VAR
  aCtrlData : ARRAY [0..9] OF WORD;
  abComp : ARRAY [0..1] OF BOOL;
  bFlag : BOOL;
  bFlagSet : BOOL;
  bFlagExe : BOOL;
  bNormal : BOOL;
  bError : BOOL;
  Mov4WORD_1 : Mov4WORD;
  iErrCode : INT;
  Mov8WORD_1 : Mov8WORD;
  Mov8WORD_2 : Mov8WORD;
  Mov8WORD_3 : Mov8WORD;
  bChange : BOOL;
  bEnableRTX : BOOL;
END_VAR
(* structured ladder/FBD written out as ST: instructions are called as NAME(EN, inputs, outputs); _pN, _eN, _tN stand for wires *)
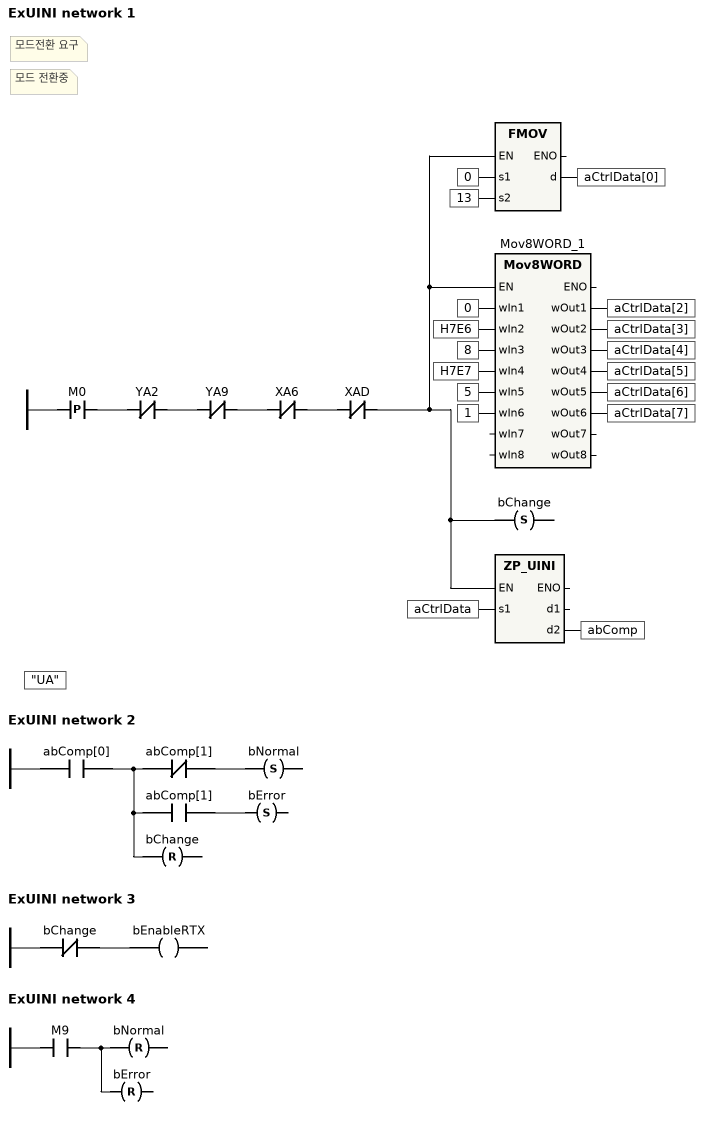
(* network 1 *)
(* 모드전환 요구 *)
(* 모드 전환중 *)
_p1 := LDP(TRUE, M0) AND NOT YA2 AND NOT YA9 AND NOT XA6 AND NOT XAD;
FMOV(_p1, 0, 13, aCtrlData[0]);
Mov8WORD_1(EN := _p1, wIn1 := 0, wIn2 := H7E6, wIn3 := 8, wIn4 := H7E7, wIn5 := 5, wIn6 := 1, wOut1 => aCtrlData[2], wOut2 => aCtrlData[3], wOut3 => aCtrlData[4], wOut4 => aCtrlData[5], wOut5 => aCtrlData[6], wOut6 => aCtrlData[7]);
ZP_UINI(_p1, aCtrlData, _open, abComp);
SET(_p1, bChange);
(* not connected to any output: "UA" *)
(* network 2 *)
SET(abComp[0] AND NOT abComp[1], bNormal);
SET(abComp[0] AND abComp[1], bError);
RST(abComp[0], bChange);
(* network 3 *)
bEnableRTX := NOT bChange;
(* network 4 *)
RST(M9, bNormal);
RST(M9, bError);
END_PROGRAM

PROGRAM ExCPRTCL_MOD
VAR
  aCtrlData : ARRAY [0..17] OF INT;
  abComp : ARRAY [0..1] OF BOOL;
  ReqFC3 : BOOL;
  Mov4INT_1 : Mov4INT;
  ReqFC5 : BOOL;
  ReqFC6 : BOOL;
  Mov4INT_2 : Mov4INT;
  Mov4INT_3 : Mov4INT;
END_VAR
(* structured ladder/FBD written out as ST: instructions are called as NAME(EN, inputs, outputs); _pN, _eN, _tN stand for wires *)
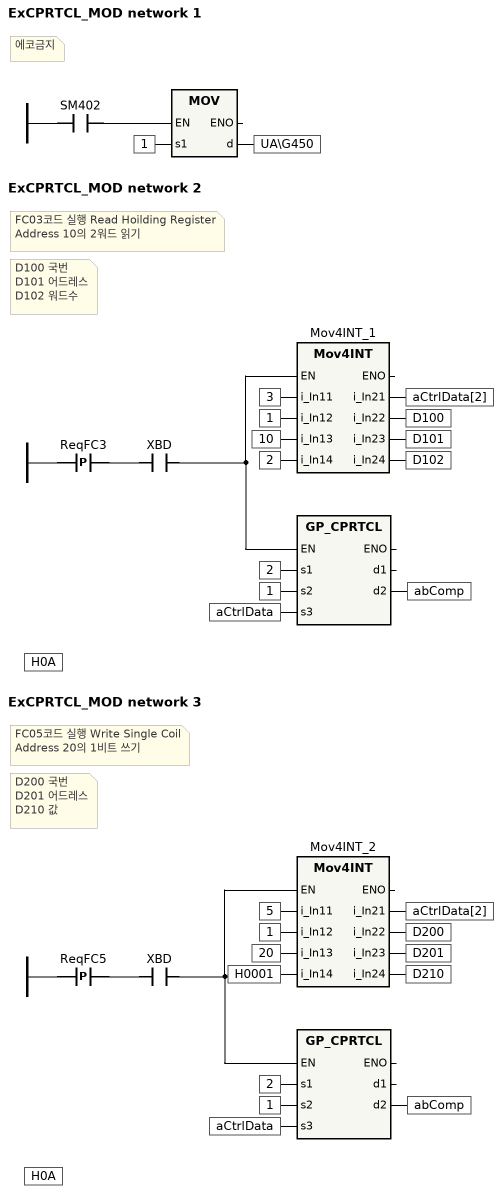
(* network 1 *)
(* 에코금지 *)
MOV(SM402, 1, UA\G450);
(* network 2 *)
(* FC03코드 실행 Read Hoilding Register  / Address 10의 2워드 읽기 *)
(* D100 국번 / D101 어드레스 / D102 워드수 *)
_p1 := LDP(TRUE, ReqFC3) AND XBD;
Mov4INT_1(EN := _p1, i_In11 := 3, i_In12 := 1, i_In13 := 10, i_In14 := 2, i_In21 => aCtrlData[2], i_In22 => D100, i_In23 => D101, i_In24 => D102);
GP_CPRTCL(_p1, 2, 1, aCtrlData, _open, abComp);
(* not connected to any output: H0A *)
(* network 3 *)
(* FC05코드 실행 Write Single Coil  / Address 20의 1비트 쓰기 *)
(* D200 국번 / D201 어드레스 / D210 값 *)
_p1 := LDP(TRUE, ReqFC5) AND XBD;
Mov4INT_2(EN := _p1, i_In11 := 5, i_In12 := 1, i_In13 := 20, i_In14 := H0001, i_In21 => aCtrlData[2], i_In22 => D200, i_In23 => D201, i_In24 => D210);
GP_CPRTCL(_p1, 2, 1, aCtrlData, _open, abComp);
(* not connected to any output: H0A *)
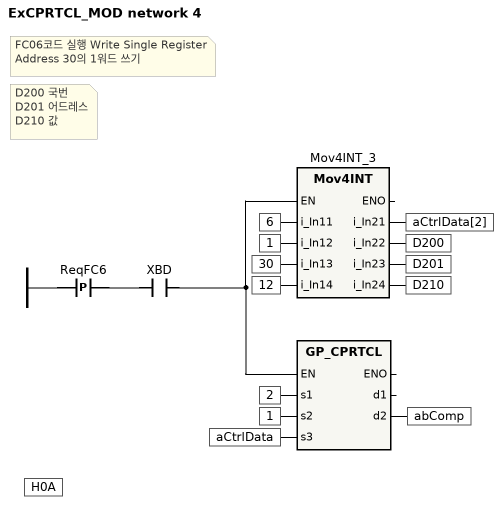
(* network 4 *)
(* FC06코드 실행 Write Single Register  / Address 30의 1워드 쓰기 *)
(* D200 국번 / D201 어드레스 / D210 값 *)
_p1 := LDP(TRUE, ReqFC6) AND XBD;
Mov4INT_3(EN := _p1, i_In11 := 6, i_In12 := 1, i_In13 := 30, i_In14 := 12, i_In21 => aCtrlData[2], i_In22 => D200, i_In23 => D201, i_In24 => D210);
GP_CPRTCL(_p1, 2, 1, aCtrlData, _open, abComp);
(* not connected to any output: H0A *)
END_PROGRAM
